INTERFACE I_PortSettings

PROPERTY PUBLIC Link : PortId
GET
END_GET
END_PROPERTY

PROPERTY PUBLIC Name : String
GET
END_GET
END_PROPERTY

PROPERTY PUBLIC PortType : String
GET
END_GET
END_PROPERTY

END_INTERFACE

(* stored: Version 1.1.0.1, ProductVersion 3.1.4024.12
   Itf I_PortSettings: Id {3c3461b8-590a-0fd1-2a86-47448a163d7b}
   Property Link: Id {ee3f220c-20b8-0bc0-039d-acde1cbf5073}
   Get Get: Id {ed2e5b85-5d77-0de4-0667-3469f1c4e80f}
   Property Name: Id {1218256f-448a-0d22-1a29-032b68480666}
   Get Get: Id {6ee9d254-3a20-0e1b-2953-9371bb00fc41}
   Property PortType: Id {82a46850-a827-0bb3-2bef-3e9ebec409e5}
   Get Get: Id {df7ac63c-33a0-0030-1bf1-c4f673474518} *)
